// TIA Portal V17 export
// export: Created 2024-09-03T21:54:55.8608831Z, ExportSetting WithDefaults, DisplayName Totally Integrated Automation Portal, DisplayVersion V17 Update 7, DisplayName TIA Portal Openness, DisplayVersion V17 Update 7, DisplayName TIA Portal Version Control Interface, DisplayVersion V17, DisplayName SINAMICS Startdrive Advanced, DisplayVersion V17 SP2, DisplayName SINAMICS Startdrive G110M, G120, G120C, G120D, G120P, G115D, DisplayVersion V17 SP2, DisplayName SINAMICS Startdrive G130, G150, S120, S150, SINAMICS MV, S210, DisplayVersion V17 SP2, DisplayName STEP 7 Professional, DisplayVersion V17 Update 7, DisplayName STEP 7 Safety, DisplayVersion V17 Update 6, DisplayName WinCC Advanced / Unified PC, DisplayVersion V17 Update 7
DATA_BLOCK "ParametersLimits_DB"   // DB40
VERSION : 0.1
// stored: AutoNumber true, DBAccessibleFromOPCUA true, DBAccessibleFromWebserver true, InstanceOfName ParametersLimits, InstanceOfType FB
"ParametersLimits"
   // VAR RETAIN
   //    limits : "udt_parametersLimits";
   // END_VAR
BEGIN
   limits.ServoPositions[0].min := 5000;
   limits.ServoPositions[1].min := 780000;
   limits.ServoPositions[2].min := 1508000;
   limits.ServoPositions[3..9].min := 0;
   limits.ServoPositions[0].max := 15000;
   limits.ServoPositions[1].max := 790000;
   limits.ServoPositions[2].max := 1518000;
   limits.ServoPositions[3..9].max := 0;
END_DATA_BLOCK
